{attribute 'qualified_only'}
VAR_GLOBAL
	GrindingWheelMS AT %Q* : BOOL;
	StartGrindingWheelPB AT %I* : BOOL;
	StopGrindingWheelPB AT %I*  : BOOL;	
END_VAR

(* stored: Version 1.1.0.1, ProductVersion 3.1.4024.4
   GVL Grinder: Id {613b322f-4b11-417d-80a3-01e55790e08f} *)
